    Pressure_Setpoint_Manual: REAL := 100.0;      // Zadane ciśnienie ręczne [bar]
    Pressure_Min_Auto       : REAL := 30.0;       // Ciśnienie startowe w auto [bar]
    Pressure_Max_Auto       : REAL := 180.0;      // Ciśnienie maksymalne w auto [bar]

    // Surowe sygnały z wejść analogowych (4-20mA)
    Raw_Position_mA         : REAL;               // np. z EL31xx
    Raw_Pressure_mA         : REAL;

    // Ustawienia sprzętowe (dostosuj pod siebie!)
    Cylinder_Stroke_mm      : REAL := 100.0;      // pełny skok siłownika [mm]
    Pressure_Sensor_Range   : REAL := 400.0;      // zakres czujnika ciśnienia [bar]

    // Parametry detekcji przebicia
    Break_Delta_Press       : REAL := 18.0;       // spadek ciśnienia [bar]
    Break_Delta_Pos         : REAL := 2.5;        // przyrost pozycji [mm]
    Break_Time_Window       : TIME := T#120ms;

    // Czas rampy ciśnienia (narastanie i opadanie)
    Ramp_Time               : TIME := T#1200MS;

END_VAR

VAR_OUTPUT
    Valve_Proportional_mA   : REAL := 4.0;        // wyjście 4-20mA do Atos
    Coil_Up                 : BOOL := FALSE;
    Coil_Down               : BOOL := FALSE;
    Valve_Relief            : BOOL := FALSE;      // odciążający – otwarty przy ruchu

    Position_mm             : REAL;              // aktualna pozycja [mm]
    Pressure_bar            : REAL;              // aktualne ciśnienie [bar]

    Auto_Running            : BOOL := FALSE;
    Breakthrough_Detected   : BOOL := FALSE;
    Press_At_Breakthrough   : REAL := 0.0;
    Pos_At_Breakthrough     : REAL := 0.0;
    Alarm                   : BOOL := FALSE;
END_VAR

VAR
    // --- wewnętrzne ---
    CycleTime_s             : REAL := 0.010;      // <-- ZMIEŃ na swój czas cyklu (0.002 = 2ms, 0.005 = 5ms itd.)

    State                   : INT := 0;           // 0=stop, 1=góra, 2=dół

    Ramp_Target_mA          : REAL := 4.0;
    Ramp_Current_mA         : REAL := 4.0;
    Ramp_Rate_mA_per_s      : REAL := 10.0;       // będzie przeliczana

    Desired_Pressure        : REAL := 0.0;

    // detekcja przebicia
    Prev_Press              : REAL := 0.0;
    Prev_Pos                : REAL := 0.0;
    Timer_Break             : TON;
    Break_Latched           : BOOL := FALSE;

    FirstCycle              : BOOL := TRUE;
END_VAR

//==========================================================================
//                        GŁÓWNA LOGIKA
//==========================================================================

// Reset przy braku Enable
IF NOT Enable THEN
    Valve_Proportional_mA := 4.0;
    Coil_Up := FALSE; Coil_Down := FALSE; Valve_Relief := FALSE;
    Auto_Running := FALSE; Alarm := FALSE; Break_Latched := FALSE;
    Breakthrough_Detected := FALSE;
    State := 0;
    Ramp_Current_mA := 4.0;
    RETURN;
END_IF;

// Skalowanie sygnałów 4-20mA → jednostki fizyczne
Position_mm  := (Raw_Position_mA  - 4.0) / 16.0 * Cylinder_Stroke_mm;
Position_mm  := LIMIT(0.0, Position_mm, Cylinder_Stroke_mm);

Pressure_bar := (Raw_Pressure_mA  - 4.0) / 16.0 * Pressure_Sensor_Range;
Pressure_bar := LIMIT(0.0, Pressure_bar, Pressure_Sensor_Range);

// Pierwsze wywołanie – zapamiętaj wartości początkowe
IF FirstCycle THEN
    Prev_Press := Pressure_bar;
    Prev_Pos   := Position_mm;
    FirstCycle := FALSE;
END_IF;

//======================================================================
// 1. Wybór trybu i komend
//======================================================================
IF Mode_Manual THEN
    // ------------------ TRYBY RĘCZNY ------------------
    Auto_Running := FALSE;
    Break_Latched := FALSE;
    Breakthrough_Detected := FALSE;

    IF Cmd_Up AND NOT Cmd_Down THEN
        State := 1;
        Desired_Pressure := GVL_HMI.nPressureSetpointManual;
		Valve_Proportional_mA := LIMIT(4.0, Ramp_Current_mA  , 20.0);
    ELSIF Cmd_Down AND NOT Cmd_Up THEN
        State := 2;
        Desired_Pressure := Pressure_Setpoint_Manual;
		Valve_Proportional_mA := LIMIT(4.0, Ramp_Current_mA  , 20.0);
    ELSE
        State := 0;
        Desired_Pressure := 0.0;
		Valve_Proportional_mA := 4.0;
    END_IF

ELSE
    // ------------------ TRYB AUTOMATYCZNY ------------------
    IF Cmd_Up AND NOT Break_Latched THEN
        Auto_Running := TRUE;
        State := 1;
		
        // ciśnienie będzie narastać od min do max wraz z pozycją
    END_IF

    IF Break_Latched THEN
        State := 0;
        Auto_Running := FALSE;
    END_IF
END_IF
IF Auto_Running THEN
	Valve_Proportional_mA := LIMIT(4.0, Ramp_Current_mA + (Pressure_Min_Auto-4), 20.0);
END_IF
//======================================================================
// 2. Sterowanie kierunkiem i zaworem odciążającym
//======================================================================
Coil_Up      := (State = 1);
Coil_Down    := (State = 2);
Valve_Relief := (State = 1) OR (State = 2);   // pompa odciążona przy każdym ruchu

//======================================================================
// 3. Oblicz docelowe ciśnienie
//======================================================================
IF Auto_Running AND State = 1 THEN
    // Narastanie ciśnienia w funkcji pozycji (mały ruch na początku → wolny wzrost)
    Desired_Pressure := Pressure_Min_Auto 
                        + (Pressure_Max_Auto - Pressure_Min_Auto); 
//                         // * (Position_mm / 60.0);        // 60 mm = pełny wzrost ciśnienia (dostosuj!)
    Desired_Pressure := LIMIT(Pressure_Min_Auto, Desired_Pressure, Pressure_Max_Auto);
END_IF;

// Przy opuszczaniu i stopie zawsze 0 bar
IF State <> 1 THEN
    Desired_Pressure := 0.0;
END_IF;

//======================================================================
// 4. Przeliczenie zadanego ciśnienia → prąd 4-20mA
//======================================================================

Ramp_Target_mA := ((Desired_Pressure+4) - Raw_Pressure_mA);

/////////Ramp_Target_mA := 4.0 + 16.0 * (Desired_Pressure / Pressure_Sensor_Range);
Ramp_Target_mA := LIMIT(4.0, Ramp_Target_mA, 20.0);

//======================================================================
// 5. Rampa ręczna (bez biblioteki)
//======================================================================
Ramp_Rate_mA_per_s := 16.0 / TIME_TO_REAL(Ramp_Time);   // ile mA na sekundę

IF Ramp_Target_mA > Ramp_Current_mA THEN
    Ramp_Current_mA := Ramp_Current_mA + Ramp_Rate_mA_per_s * CycleTime_s;
    IF Ramp_Current_mA > Ramp_Target_mA THEN Ramp_Current_mA := Ramp_Target_mA; END_IF;
ELSIF Ramp_Target_mA < Ramp_Current_mA THEN
    Ramp_Current_mA := Ramp_Current_mA - Ramp_Rate_mA_per_s * CycleTime_s;
    IF Ramp_Current_mA < Ramp_Target_mA THEN Ramp_Current_mA := Ramp_Target_mA; END_IF;
END_IF;

// Valve_Proportional_mA := LIMIT(4.0, Ramp_Current_mA + Pressure_Min_Auto, 20.0);

//======================================================================
// 6. Detekcja przebicia materiału
//======================================================================
IF State = 1 THEN
    IF (Prev_Press - Pressure_bar) > Break_Delta_Press 
       AND (Position_mm - Prev_Pos) > Break_Delta_Pos THEN
        Timer_Break(IN := TRUE, PT := Break_Time_Window);
        IF Timer_Break.Q THEN
            Break_Latched         := TRUE;
            Breakthrough_Detected := TRUE;
            Press_At_Breakthrough := Pressure_bar;
            Pos_At_Breakthrough   := Position_mm;
            Alarm                 := TRUE;
        END_IF
    ELSE
        Timer_Break(IN := FALSE);
    END_IF
ELSE
    Timer_Break(IN := FALSE);
END_IF

//======================================================================
// 7. Zatrzymanie po przebiciu
//======================================================================
IF Break_Latched THEN
    State := 0;
    Valve_Proportional_mA := 4.0;   // natychmiast zamknięty
END_IF

// Zapamiętaj wartości na następny cykl
Prev_Press := Pressure_bar;
Prev_Pos   := Position_mm;

END_FUNCTION_BLOCK

// ---- POUs/POUs/Recipe/RecipeManagement.TcPOU
PROGRAM RecipeManagement
VAR
	bInit					: BOOL := TRUE;
	fbRecipeManComm			: RecipeManCommands;
	sRecipeDef				: STRING := 'Recipes';
	nCount					: INT;
	nPreviousSelectionIndex	: INT := -2;
	nLastError				: DWORD;
	nRecipeCount			: INT;
	nPreviousIndex			: INT;
	bReloadValues			: BOOL;
	nSelectionIndexInList 	: INT;
	sRecipe					: STRING;
	bReload					: BOOL;
	bSave					: BOOL;
	sNewRecipeName			: STRING;
	bSaveVariables			: BOOL;
	fbSaveVariablesTrigger	: R_TRIG;
	sLoadName				: STRING;
	fbLoadTrigger			: R_TRIG;
	bDelete					: BOOL;
	bCreate					: BOOL;
	bSaveHMI				: BOOL;
	ftRefresh				: F_TRIG;
	tp1						: TP;
	sHmi_Name				: STRING;
	i: INT;
	j: INT;
	iKrokTryb: INT;
	bRecipeToPLC: BOOL;
	arrPusty: ARRAY[0..30] OF INT;
END_VAR




GVL_HMI.uiIloscReceptur:=INT_TO_UINT(GVL_Recipe.nRecipeCount-1);
A_ReadRecipe();
// inicjalizacjia
tp1(In:=bDelete OR bCreate OR bSaveHMI, PT:=T#100MS);
ftRefresh(CLK:=tp1.Q);
IF ftRefresh.Q THEN
	bReload:=TRUE;
END_IF
IF bInit THEN
	// pobierz liczbe receptur
	GVL_Recipe.nRecipeCount:=fbRecipeManComm.GetRecipeCount(sRecipeDef);
	// wyczysc wszystkie tablice
	FOR nCount := 0 TO GVL_Recipe.cMaxTableRows DO
		GVL_Recipe.aRecipeNames[nCount] := '';
		//GVL_Recipe.aVariableNames[nCount] := '';
		GVL_Recipe.aVariableValues[nCount] := '';
	END_FOR
	
	fbRecipeManComm.GetRecipeNames(sRecipeDef,
									ADR(GVL_Recipe.aRecipeNames),
									30,
									GVL_Recipe.nRecipeIndex);
										
	GVL_Recipe.nRecipeSelectionIndex := -1;
	nPreviousSelectionIndex := -1;
	bInit := FALSE;
END_IF

nRecipeCount := fbRecipeManComm.GetRecipeCount(sRecipeDef);
nLastError := fbRecipeManComm.GetLastError();


// scroll position has changed
IF GVL_Recipe.nRecipeIndex <> nPreviousIndex THEN
	fbRecipeManComm.GetRecipeNames(	sRecipeDef,
									ADR(GVL_Recipe.aRecipeNames),
									30,
									GVL_Recipe.nRecipeIndex);
	nPreviousIndex := GVL_Recipe.nRecipeIndex;
END_IF


//============================================================================
CASE iKrokTryb OF
	0:IF bRecipeToPLC THEN
		iKrokTryb:=10;
	END_IF
	10:
	GVL_Recipe.nRecipeSelectionIndexTemp:=GVL_Recipe.nRecipeSelectionIndex;
	iKrokTryb:=20;
	bRecipeToPLC:=FALSE;
	20:
	GVL_Recipe.nRecipeSelectionIndex:=0;
fbRecipeManComm.ReloadRecipes(sRecipeDef);
	
	iKrokTryb:=25;
	25:
	GVL_Recipe.nRecipeSelectionIndex:=30;
	iKrokTryb:=30;
	30:
	GVL_Recipe.nRecipeSelectionIndex:=GVL_Recipe.nRecipeSelectionIndexTemp;
	iKrokTryb:=40;
	40:
	fbRecipeManComm.WriteRecipe(sRecipeDef,sRecipe);
	iKrokTryb:=0;
END_CASE



//==========================================================


//selection changed
IF GVL_Recipe.nRecipeSelectionIndex <> nPreviousSelectionIndex OR bReloadValues THEN
	nPreviousSelectionIndex := GVL_Recipe.nRecipeSelectionIndex;
	nSelectionIndexInList := GVL_Recipe.nRecipeSelectionIndex - GVL_Recipe.nRecipeIndex;
	
	(* Get the selected recipe name *)
	IF nSelectionIndexInList >= 0 AND nSelectionIndexInList < 30 THEN
		sRecipe := GVL_Recipe.aRecipeNames[nSelectionIndexInList];
	END_IF
	
	fbRecipeManComm.GetRecipeVariableNames(sRecipeDef, sRecipe,ADR(GVL_Recipe.aVariableNames),30,0);
	
	fbRecipeManComm.GetRecipeValues(sRecipeDef,
										sRecipe,
										ADR(GVL_Recipe.aVariableValues),
										30,
										GVL_Recipe.nVariableIndex,
										80);
										
(*	fbRecipeManComm.GetRecipeVariableNames(	sRecipeDef,
												sRecipe,
												ADR(GVL_Recipe.aVariableNames),
												10,
												GVL_Recipe.nVariableIndex);*)
	
	bReloadValues := FALSE;
END_IF
	
IF bReload THEN
	fbRecipeManComm.ReloadRecipes(sRecipeDef);
	bInit := TRUE;
	bReload := FALSE;
END_IF

fbSaveVariablesTrigger(CLK := bSaveVariables);
IF fbSaveVariablesTrigger.Q THEN
	fbRecipeManComm.SetRecipeValues(sRecipeDef,
									sRecipe,
									ADR(GVL_Recipe.aVariableValues),
									30,
									GVL_Recipe.nVariableIndex);	
	bSaveVariables := FALSE;
END_IF

IF bSave THEN
	fbRecipeManComm.SaveRecipe(sRecipeDef, sRecipe);
	bSave:=FALSE;
END_IF

bReload := FALSE;
sHmi_Name:=CONCAT(str1:=(CONCAT(str1:=sRecipeDef,str2:=' ')),str2:=sRecipe);

ACTION A_ReadRecipe:
GVL_Recipe.aCurrentValues[0]:=BreakthroughDetection.nBreakDeltaPos;
GVL_Recipe.aCurrentValues[1]:=arrPusty[1];;
GVL_Recipe.aCurrentValues[2]:=arrPusty[1];;
GVL_Recipe.aCurrentValues[3]:=arrPusty[1];;
GVL_Recipe.aCurrentValues[4]:=arrPusty[1];;
GVL_Recipe.aCurrentValues[5]:=arrPusty[1];;
GVL_Recipe.aCurrentValues[6]:=arrPusty[1];;
GVL_Recipe.aCurrentValues[7]:=arrPusty[1];;
GVL_Recipe.aCurrentValues[8]:=arrPusty[1];;
GVL_Recipe.aCurrentValues[9]:=arrPusty[1];;
GVL_Recipe.aCurrentValues[10]:=arrPusty[1];;
GVL_Recipe.aCurrentValues[11]:=arrPusty[1];
GVL_Recipe.aCurrentValues[12]:=arrPusty[2];
GVL_Recipe.aCurrentValues[13]:=arrPusty[3];
GVL_Recipe.aCurrentValues[14]:=arrPusty[4];
END_ACTION

END_PROGRAM

// ---- GlobalTextList.TcGTLO
TEXTLIST GlobalTextList
  903 = ''
  81 = '\t\tz'
  895 = ' Odczyt pozycji'
  846 = '%'
  355 = '%.1f'
  987 = '%.2f'
  26 = '%.2F'
  546 = '%i'
  346 = '%s'
  974 = '%S'
  1490 = '%t[mm.ss] min'
  312 = '2'
  76 = 'Admin'
  462 = 'Aktualna receptura:'
  378 = 'ALARMY'
  845 = 'bar'
  210 = 'Ciśnienie'
  83 = 'Ciśnienie przebicia'
  981 = 'Ciśnienie przebicia:  %.2f'
  144 = 'Ciśnienie przebicia:  %.2f [bar]'
  195 = 'Ciśnienie przebicia:%.2f'
  658 = 'Ciśnienie:  %.2f [bar]'
  430 = 'Czas narastania ciśnienia:  %i [ms]'
  959 = 'Czas narastania ciśnienia:  %i [s]'
  190 = 'Czas start'
  191 = 'Czas stop'
  838 = 'GŁÓWNY'
  851 = 'Ilość receptur'
  825 = 'MAIN'
  824 = 'Nastawa ciśnienia'
  373 = 'Nastawa ciśnienia-AUTO-Max:  %.2f [bar]'
  919 = 'Nastawa ciśnienia-AUTO-Min:  %.2f [bar]'
  526 = 'Nastawa ciśnienia-AUTO:  %.2f'
  415 = 'Nastawa ciśnienia-AUTO:  %.2f [bar]'
  790 = 'Nastawa ciśnienia-AUTO:%.2f'
  523 = 'Nastawa ciśnienia-RĘKA:  %.2f [bar]'
  442 = 'Nastawa ciśnienia-Ręka:  %.2f [bar]'
  570 = 'Nastawa ciśnienia-RĘKA:%.2f'
  705 = 'Nastawa ciśnienia:%.2f'
  404 = 'Nazwa nowej receptury'
  169 = 'Nazwa zmiennej'
  171 = 'Odczyt ciśnienia'
  49 = 'Odczyt ciśnienia:  %.2f'
  360 = 'Odczyt ciśnienia:  %.2f [bar]'
  365 = 'Odczyt ciśnienia:%.2f'
  107 = 'Odczyt pozycji:  %.2f'
  429 = 'Odczyt pozycji:  %.2f [mm]'
  129 = 'Odczyt pozycji:%.2f'
  173 = 'Okno czasowe:  %.2f [bar]'
  474 = 'Okno czasowe:  %.2f [ms]'
  10 = 'Okno czasowe:  %i [ms]'
  627 = 'Operator'
  823 = 'PLC -> \nReceptura'
  193 = 'Pozycja przebicia'
  498 = 'Pozycja przebicia:  %.2f'
  375 = 'Pozycja przebicia:  %.2f [mm]'
  387 = 'Pozycja przebicia:%.2f'
  126 = 'Pozycja startowa:  %.2f [mm]'
  286 = 'Pozycja:  %.2f [mm]'
  535 = 'Recptura ->\n PLC'
  468 = 'RESET'
  247 = 'RESET\nCYKLU  >5s'
  1191 = 'RESET\nŻĄDANIA\nPŁUKANIA'
  431 = 'Service'
  622 = 'Siła (p*A):  %.2f [kN]'
  818 = 'Siła przebicia:  %.2f [bar]'
  639 = 'Siła przebicia:  %.2f [kN]'
  731 = 'Siła przebicia:  %.2f [tf]'
  235 = 'Siła(p*A):  %.2f [tf]'
  887 = 'Siła:  %.2f [bar]'
  22 = 'Siła:  %.2f [kg]'
  99 = 'Siła:  %.2f [kN]'
  989 = 'Siła:  %.2f [N]'
  496 = 'Siła:  %.2f [tf]'
  576 = 'Siła:  %.2f [t]'
  563 = 'Spadek ciśnienia:  %.2f [bar]'
  178 = 'TYLKO\nAKTYWNE'
  200 = 'USTAWIENIA'
  789 = 'Usuń wybraną\n recepturę'
  500 = 'Utwórz nową recepturę \nz wartościami PLC'
  396 = 'Wartość z plc'
  847 = 'Wartość z receptury'
  172 = 'WYBÓR\nRECEPTURY'
  447 = 'Wzrost pozycji:  %.2f [bar]'
  319 = 'Wzrost pozycji:  %.2f [mm]'
  57 = 'ZAKRES TENSOMETRU'
  638 = 'Zapisz wybraną \nrecepturę \ndo pliku'
  1546 = 'ZARZĄDZANIE \nUŻYTKOWNIKAMI'
  727 = 'Zastosuj zmiany'
  952 = 'ZATWIERDŹ'
  933 = 'Załaduj z pliku\n i wpisz do PLC'
  876 = 'ZEROWANIE\n POZYCJI TŁOKA'
  772 = 'Zerowanie pozycji'
END_TEXTLIST

// ---- HMI/ListyTextowe/PrzyciskAlarmy.TcTLO
TEXTLIST PrzyciskAlarmy
  1 = 'AKTYWNE'
  0 = 'WSZYSTKIE'
   = ''
END_TEXTLIST

// ---- HMI/ListyTextowe/Tensometr.TcTLO
TEXTLIST Tensometr
  0 = '50t'
  1 = '100t'
   = ''
END_TEXTLIST

// ---- HMI/ListyTextowe/TextList_Przyciski_Menu.TcTLO
TEXTLIST TextList_Przyciski_Menu
  0 = 'GŁÓWNA'
  1 = 'ALARMY'
  2 = 'USTAWIENIA'
   = ''
END_TEXTLIST

// ---- HMI/NEW_VISU/Frames/E0.TcVIS
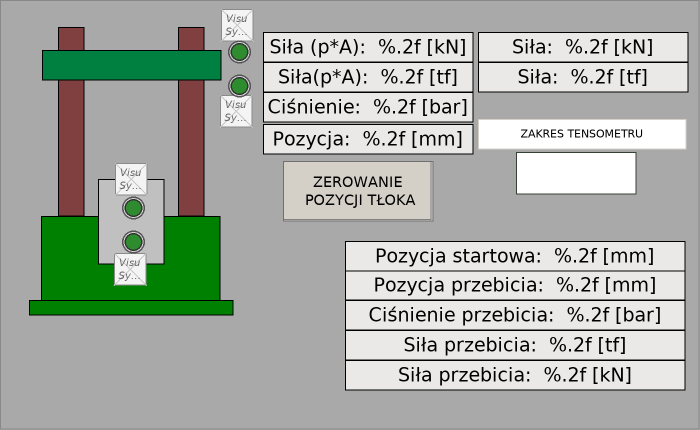
VISUALIZATION E0  // 700x430
    Textfield (263,92 210x30), "Ciśnienie: %.2f [bar]", text variable: Scaling.PressureAI.PV_Value
    Textfield (263,124 210x30), "Pozycja: %.2f [mm]", text variable: Scaling.fbPos.PosZeroed_mm
    Textfield (345,300 340x30), "Ciśnienie przebicia: %.2f [bar]", text variable: GVL_HMI.nPressBreak
    Textfield (345,270 340x30), "Pozycja przebicia: %.2f [mm]", text variable: GVL_HMI.nPositionBreak
    Textfield (345,241 340x30), "Pozycja startowa: %.2f [mm]", text variable: GVL_HMI.nPositionStart
    Rectangle (58,27 26x189)
    Rectangle (178,27 26x189)
    Rectangle (41,216 179x85)
    Rectangle (98,179 66x85)
    Rectangle (42,50 179x30)
    Group (220,9 35x118)
        Group (1,0 34x56)
            Image (0,0 32x32), colour toggle: bTopPreserUp, image: VisuSymbols.Symbols.ArrowBoldUp
            Lamp1 (3,30 31x26), variable: bTopPreserDown, style: Lamp-Lamp1-Green
        Group (0,64 35x54)
            Image (0,22 32x32), image: VisuSymbols.Symbols.ArrowBoldDown
            Lamp1 (4,0 31x26), variable: bTopPreserUp, style: Lamp-Lamp1-Green
    Group (114,163 35x122)
        Group (1,0 34x58)
            Image (0,0 32x32), colour toggle: bCylinderValveUp, image: VisuSymbols.Symbols.ArrowBoldUp
            Lamp1 (3,32 31x26), variable: bCylinderValveUp, style: Lamp-Lamp1-Green
        Group (0,66 35x56)
            Image (0,24 32x32), colour toggle: bCylinderValveDown, image: VisuSymbols.Symbols.ArrowBoldDown
            Lamp1 (4,0 31x26), variable: bCylinderValveDown, style: Lamp-Lamp1-Green
    Textfield (263,62 210x30), "Siła(p*A): %.2f [tf]", text variable: GVL_HMI.Force_kg/1000
    Textfield (263,32 210x30), "Siła (p*A): %.2f [kN]", text variable: GVL_HMI.Force_N/1000
    Rectangle (29,300 204x15)
    Textfield (478,62 210x30), "Siła: %.2f [tf]", text variable: GVL_ForceMode.nForce_t
    Textfield (478,32 210x30), "Siła: %.2f [kN]", text variable: GVL_ForceMode.nForce_kN
    Rectangle (516,152 120x42), colour toggle: P_EventsVisu.bFilterActiveOnly, input disabled if: bLedCycleOn, text list: 'Tensometr', text index: GVL_ForceMode.bForceRange100t
        toggle GVL_ForceMode.bForceRange100t
    Textfield (345,330 340x30), "Siła przebicia: %.2f [tf]", text variable: GVL_HMI.nForce_t_Break
    Textfield (345,360 340x30), "Siła przebicia: %.2f [kN]", text variable: GVL_HMI.nForce_kN_Break
    Textfield (478,119 208x30), "ZAKRES TENSOMETRU"
    Button (283,161 150x60), "ZEROWANIE POZYCJI TŁOKA", input disabled if: bLedCycleOn
        OnMouseDown: execute { Scaling.fbPos.SetZero:=false; }
        OnMouseUp: execute { Scaling.fbPos.SetZero:=true; }
END_VISUALIZATION

// ---- HMI/NEW_VISU/Frames/E1.TcVIS
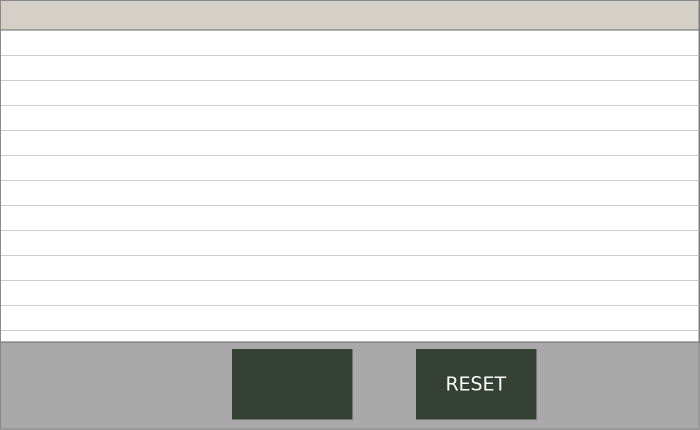
VISUALIZATION E1  // 700x430
    Table (0,0 700x342), data array: GVL_EHS.arrEventVisu
        p3854506369: GVL_EHS.arrEventVisu[INDEX].dwID
        p1892666644: GVL_EHS.arrEventVisu[INDEX].dwParam
        p1218418051: GVL_EHS.arrEventVisu[INDEX].wsMessage
        p746581629: GVL_EHS.arrEventVisu[INDEX].dwColor
        p511219082: Class
        p505689113: Czas ustąpienia
        p3312258591: GVL_EHS.arrEventVisu[INDEX].dwClass
        p2340480326: GVL_EHS.arrEventVisu[INDEX].dtDateEnd
        p1755163831: Opis zdarzenia
        p2237128397: Czas stop
        p2170511999: GVL_EHS.arrEventVisu[INDEX].dtDateBegin
        p4092479075: Czas start
    Rectangle (416,349 120x70), "RESET", colour toggle: GVL_HMI.bResetAlarm
        OnMouseDown: execute { GVL_HMI.bResetAlarm:=TRUE; }
        OnMouseUp: execute { GVL_HMI.bResetAlarm:=FALSE; }
    Rectangle (232,349 120x70), colour toggle: P_EventsVisu.bFilterActiveOnly, text list: 'PrzyciskAlarmy', text index: P_EventsVisu.bFilterActiveOnly
        toggle P_EventsVisu.bFilterActiveOnly
END_VISUALIZATION

// ---- HMI/NEW_VISU/Frames/E2.TcVIS
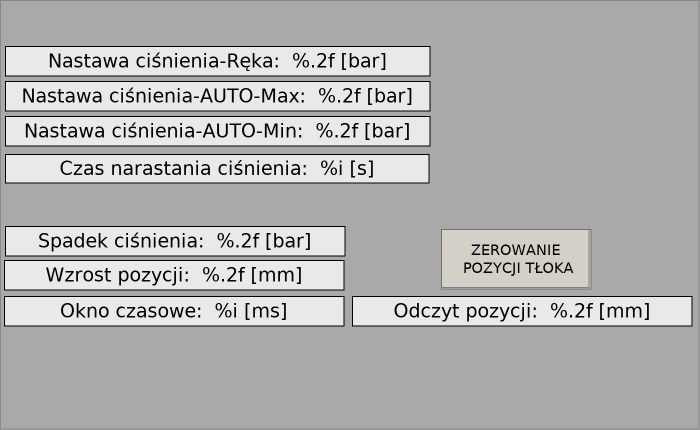
VISUALIZATION E2  // 700x430
    Textfield (5,81 425x30), "Nastawa ciśnienia-AUTO-Max: %.2f [bar]", text variable: GVL_HMI.PressureSetpointAutoMax
        OnMouseDown: write the text variable via Default, min 0, max 300
    Textfield (5,46 425x30), "Nastawa ciśnienia-Ręka: %.2f [bar]", text variable: GVL_HMI.nPressureSetpointManual
        OnMouseDown: write the text variable via Default, min 0, max 200
    Textfield (5,116 425x30), "Nastawa ciśnienia-AUTO-Min: %.2f [bar]", text variable: GVL_HMI.PressureSetpointAutoMin
        OnMouseDown: write the text variable via Default, min 0, max 300
    Textfield (5,226 340x30), "Spadek ciśnienia: %.2f [bar]", text variable: GVL_HMI.nBreakDeltaPress
        OnMouseDown: write the text variable via Default, min 0, max 200
    Textfield (4,260 340x30), "Wzrost pozycji: %.2f [mm]", text variable: GVL_HMI.nBreakDeltaPos
        OnMouseDown: write the text variable via Default, min 0, max 200
    Textfield (4,296 340x30), "Okno czasowe: %i [ms]", text variable: GVL_HMI.nBreak_Time_Window
        OnMouseDown: write the text variable via Default, min 0, max 200
    Textfield (5,154 424x29), "Czas narastania ciśnienia: %i [s]", text variable: GVL_HMI.nRamp_Time
        OnMouseDown: write the text variable via Default, min 0, max 3600
    Textfield (352,296 340x30), "Odczyt pozycji: %.2f [mm]", text variable: Scaling.fbPos.PosZeroed_mm
    Button (441,229 150x60), "ZEROWANIE POZYCJI TŁOKA", input disabled if: bLedCycleOn
        OnMouseDown: execute { Scaling.fbPos.SetZero:=false; }
        OnMouseUp: execute { Scaling.fbPos.SetZero:=true; }
END_VISUALIZATION

// ---- HMI/NEW_VISU/MAIN.TcVIS
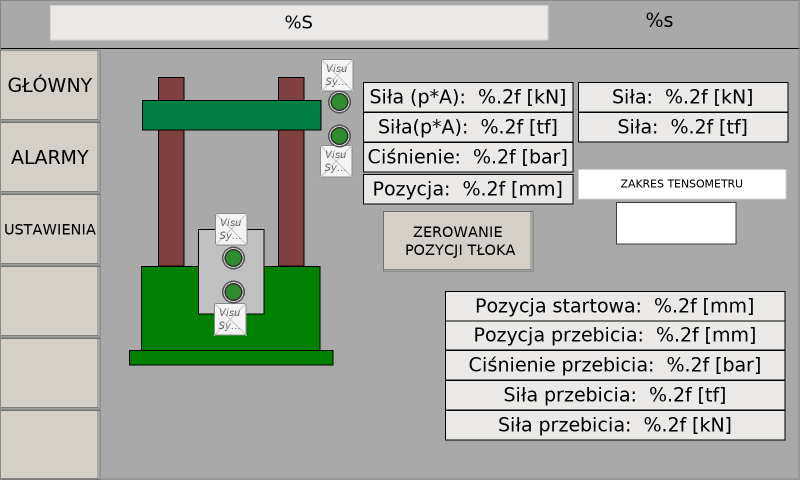
VISUALIZATION MAIN  // 800x480
    Frame (100,50 700x430)
        shows E0()
        shows E1()
        shows E2()
    Frame (0,50 100x430)
        shows MENU_2()
    Frame (0,0 800x50)
        shows TOP()
        shows MENU_2()
END_VISUALIZATION

// ---- HMI/NEW_VISU/MENU_2.TcVIS
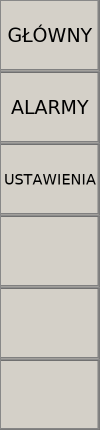
VISUALIZATION MENU_2  // 100x430
    Button (0,0 100x71), "GŁÓWNY", colour toggle: GVL_HMI.hmiPanel.uiNumerEkranu=0
        OnMouseUp: FrameSelectionChange Selection=Selection=-1, GlobSel=IndExpr=0, AssignDir=MAIN.Frames, AssignType=Directly, SelType=Globally
        OnMouseUp: execute { GVL_HMI.hmiPanel.uiMenu	 :=0; GVL_HMI.hmiPanel.bResetMenu := TRUE; }
    Button (0,72 100x71), "ALARMY", colour toggle: GVL_HMI.hmiPanel.uiNumerEkranu=1
        OnMouseUp: FrameSelectionChange Selection=Selection=-1, GlobSel=IndExpr=1, AssignDir=MAIN.Frames, AssignType=Directly, SelType=Globally
        OnMouseUp: execute { GVL_HMI.hmiPanel.uiMenu	 :=1; GVL_HMI.hmiPanel.bResetMenu := TRUE; }
    Button (0,216 100x71)
    Button (0,288 100x71)
    Button (0,360 100x70)
    Button (0,144 100x71), "USTAWIENIA", colour toggle: GVL_HMI.hmiPanel.uiNumerEkranu=2
        OnMouseUp: FrameSelectionChange Selection=Selection=-1, GlobSel=IndExpr=2, AssignDir=MAIN.Frames, AssignType=Directly, SelType=Globally
        OnMouseUp: execute {
            GVL_HMI.hmiPanel.uiMenu	 :=2
            ;
            GVL_HMI.hmiPanel.bResetMenu := TRUE;
        }
END_VISUALIZATION

// ---- HMI/NEW_VISU/TOP.TcVIS
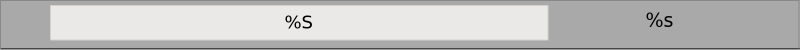
VISUALIZATION TOP  // 800x50
    Line (0,48) (800,48)
    Textfield (526,1 267x39), "%s", text variable: GVL_EHS.dtActTime
    Textfield (50,5 498x35), "%S", text variable: GVL_HMI.sMode
END_VISUALIZATION
